(* Logix 5000 project; controller Amvex_Thorpe_Flowmeter vendor 1 type 14 code 106 rev 33.13; software revision 33.01; part 15 of 16 *)
(* tags used below, declared in another part *)
   Auto_Seq : SEQ;
   Clear_TM : TIMER;
   Counter_ONS : BOOL;
   FAULT : DINT;
   FAULTED : DINT;
   Flash_Timer_Off : TIMER;
   Flash_Timer_On : TIMER;
   MODE : MODE;
   RCD_ONS : BOOL;
   RESET : BOOL;
   RESET_ONS : BOOL;
   End_Of_Cycle : BOOL;
   Fitting_Cycle_Timer : TIMER;
   Fitting_Cycle_Timer_DINT : DINT;
   Fitting_Cycle_Timer_ONS : BOOL;
   HMI : HMI_Temp;
   RCP1 : RCP1;
   RCP1_00 : UDT_ID0;
(* RPC1_Main, continued *)

ROUTINE R02_OUTPUTS   (* ladder *)
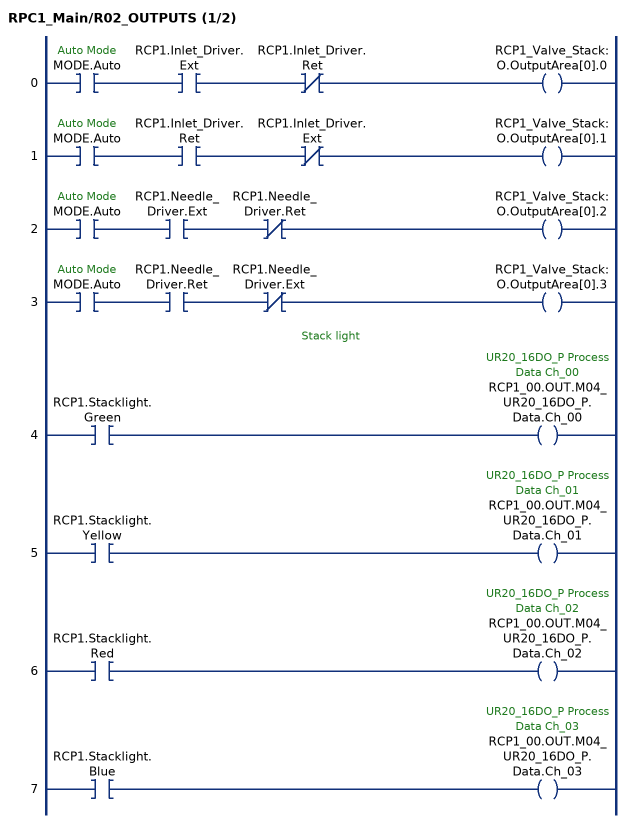
   0: XIC(MODE.Auto)XIC(RCP1.Inlet_Driver.Ext)XIO(RCP1.Inlet_Driver.Ret)OTE(RCP1_Valve_Stack:O.OutputArea[0].0);
   1: XIC(MODE.Auto)XIC(RCP1.Inlet_Driver.Ret)XIO(RCP1.Inlet_Driver.Ext)OTE(RCP1_Valve_Stack:O.OutputArea[0].1);
   2: XIC(MODE.Auto)XIC(RCP1.Needle_Driver.Ext)XIO(RCP1.Needle_Driver.Ret)OTE(RCP1_Valve_Stack:O.OutputArea[0].2);
   3: XIC(MODE.Auto)XIC(RCP1.Needle_Driver.Ret)XIO(RCP1.Needle_Driver.Ext)OTE(RCP1_Valve_Stack:O.OutputArea[0].3);
   // Stack light
   4: XIC(RCP1.Stacklight.Green)OTE(RCP1_00.OUT.M04_UR20_16DO_P.Data.Ch_00);
   5: XIC(RCP1.Stacklight.Yellow)OTE(RCP1_00.OUT.M04_UR20_16DO_P.Data.Ch_01);
   6: XIC(RCP1.Stacklight.Red)OTE(RCP1_00.OUT.M04_UR20_16DO_P.Data.Ch_02);
   7: XIC(RCP1.Stacklight.Blue)OTE(RCP1_00.OUT.M04_UR20_16DO_P.Data.Ch_03);
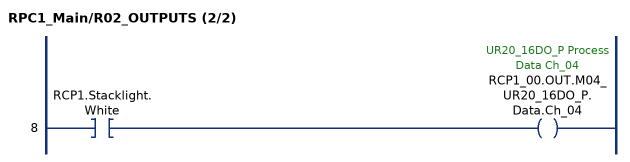
   8: XIC(RCP1.Stacklight.White)OTE(RCP1_00.OUT.M04_UR20_16DO_P.Data.Ch_04);
END_ROUTINE

ROUTINE R03_AUTO_SEQ   (* ladder *)
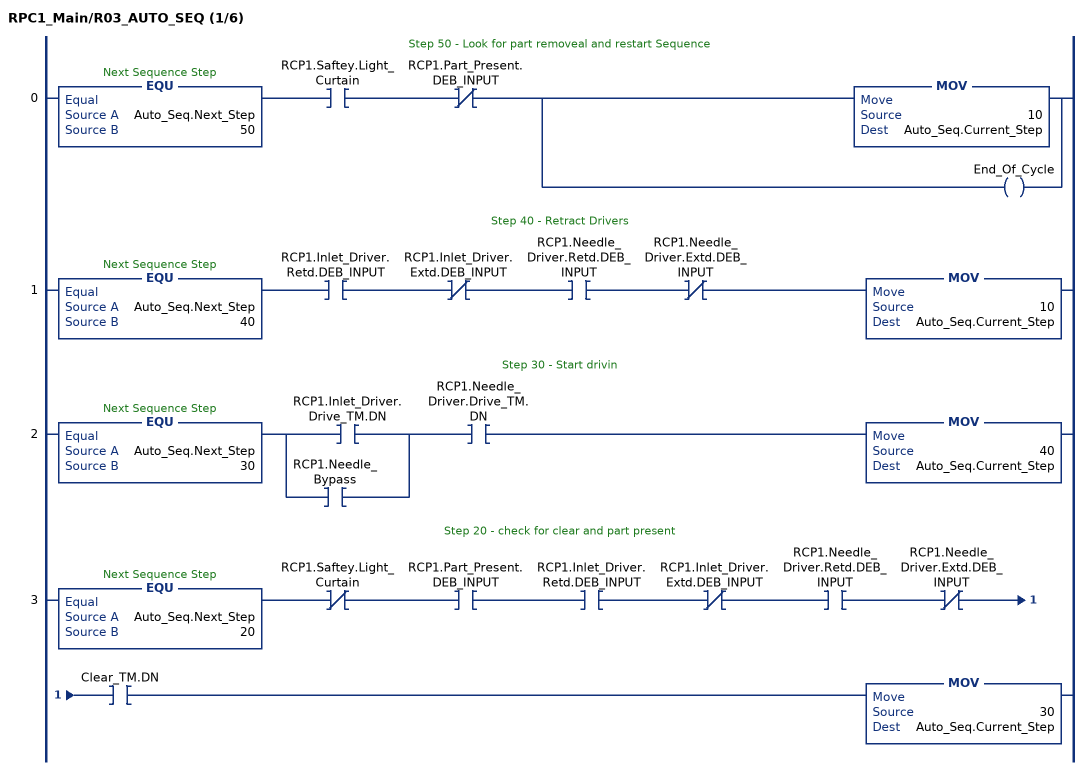
   // Step 50 - Look for part removeal and restart Sequence
   0: EQU(Auto_Seq.Next_Step,50)XIC(RCP1.Saftey.Light_Curtain)XIO(RCP1.Part_Present.DEB_INPUT)[MOV(10,Auto_Seq.Current_Step) ,OTE(End_Of_Cycle) ];
   // Step 40 - Retract Drivers
   1: EQU(Auto_Seq.Next_Step,40)XIC(RCP1.Inlet_Driver.Retd.DEB_INPUT)XIO(RCP1.Inlet_Driver.Extd.DEB_INPUT)XIC(RCP1.Needle_Driver.Retd.DEB_INPUT)XIO(RCP1.Needle_Driver.Extd.DEB_INPUT)MOV(10,Auto_Seq.Current_Step);
   // Step 30 - Start drivin
   2: EQU(Auto_Seq.Next_Step,30)[XIC(RCP1.Inlet_Driver.Drive_TM.DN) ,XIC(RCP1.Needle_Bypass) ]XIC(RCP1.Needle_Driver.Drive_TM.DN)MOV(40,Auto_Seq.Current_Step);
   // Step 20 - check for clear and part present
   3: EQU(Auto_Seq.Next_Step,20)XIO(RCP1.Saftey.Light_Curtain)XIC(RCP1.Part_Present.DEB_INPUT)XIC(RCP1.Inlet_Driver.Retd.DEB_INPUT)XIO(RCP1.Inlet_Driver.Extd.DEB_INPUT)XIC(RCP1.Needle_Driver.Retd.DEB_INPUT)XIO(RCP1.Needle_Driver.Extd.DEB_INPUT)XIC(Clear_TM.DN)MOV(30,Auto_Seq.Current_Step);
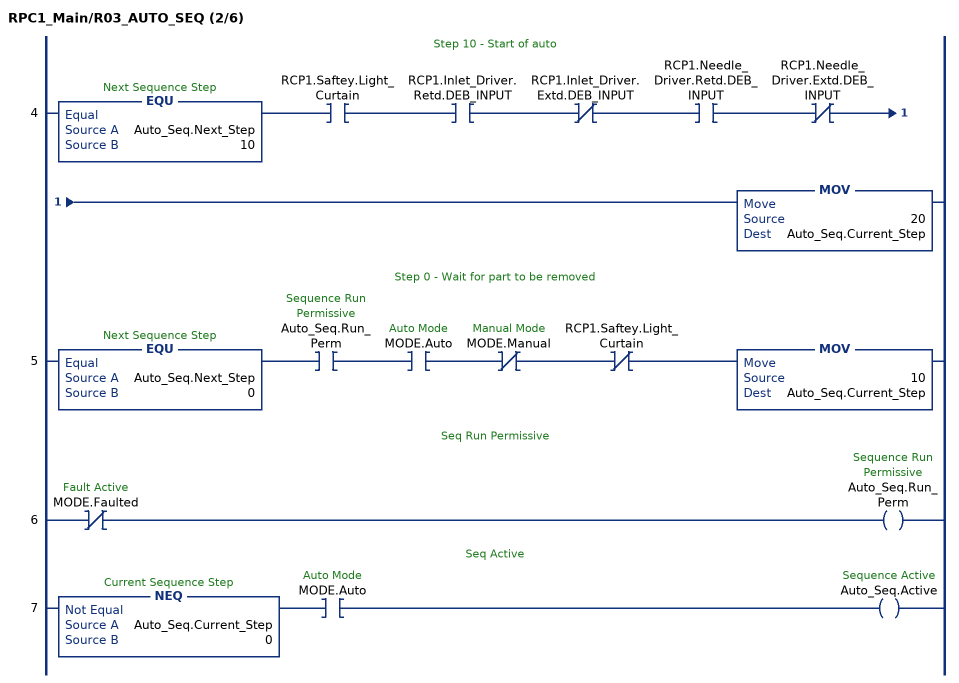
   // Step 10 - Start of auto
   4: EQU(Auto_Seq.Next_Step,10)XIC(RCP1.Saftey.Light_Curtain)XIC(RCP1.Inlet_Driver.Retd.DEB_INPUT)XIO(RCP1.Inlet_Driver.Extd.DEB_INPUT)XIC(RCP1.Needle_Driver.Retd.DEB_INPUT)XIO(RCP1.Needle_Driver.Extd.DEB_INPUT)MOV(20,Auto_Seq.Current_Step);
   // Step 0 - Wait for part to be removed
   5: EQU(Auto_Seq.Next_Step,0)XIC(Auto_Seq.Run_Perm)XIC(MODE.Auto)XIO(MODE.Manual)XIO(RCP1.Saftey.Light_Curtain)MOV(10,Auto_Seq.Current_Step);
   // Seq Run Permissive
   6: XIO(MODE.Faulted)OTE(Auto_Seq.Run_Perm);
   // Seq Active
   7: NEQ(Auto_Seq.Current_Step,0)XIC(MODE.Auto)OTE(Auto_Seq.Active);
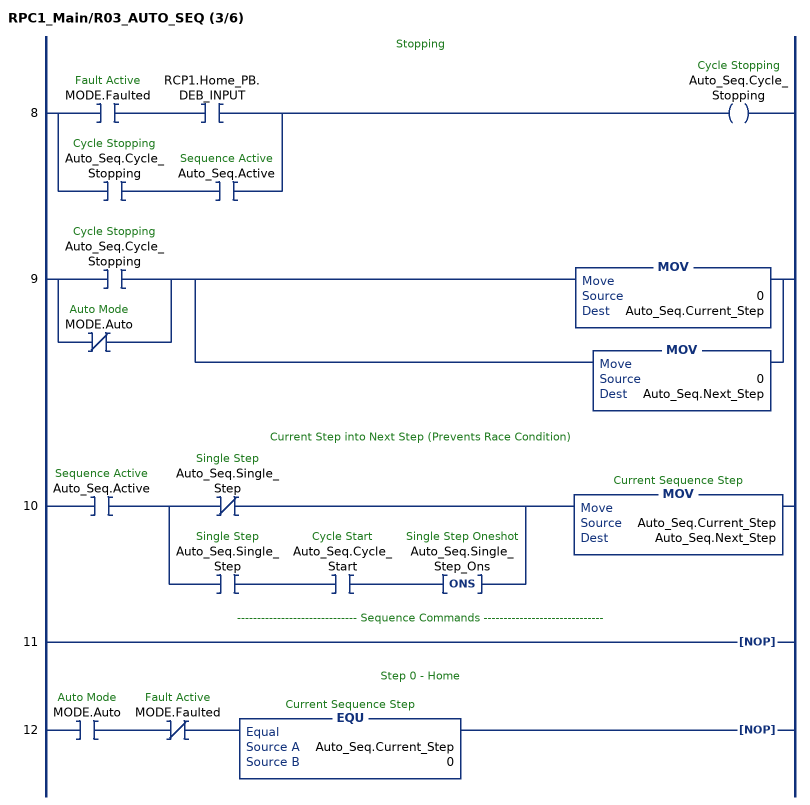
   // Stopping
   8: [XIC(MODE.Faulted) XIC(RCP1.Home_PB.DEB_INPUT) ,XIC(Auto_Seq.Cycle_Stopping) XIC(Auto_Seq.Active) ]OTE(Auto_Seq.Cycle_Stopping);
   9: [XIC(Auto_Seq.Cycle_Stopping) ,XIO(MODE.Auto) ][MOV(0,Auto_Seq.Current_Step) ,MOV(0,Auto_Seq.Next_Step) ];
   // Current Step into Next Step (Prevents Race Condition)
   10: XIC(Auto_Seq.Active)[XIO(Auto_Seq.Single_Step) ,XIC(Auto_Seq.Single_Step) XIC(Auto_Seq.Cycle_Start) ONS(Auto_Seq.Single_Step_Ons) ]MOV(Auto_Seq.Current_Step,Auto_Seq.Next_Step);
   // ------------------------------ Sequence Commands ------------------------------
   11: NOP();
   // Step 0 - Home
   12: XIC(MODE.Auto)XIO(MODE.Faulted)EQU(Auto_Seq.Current_Step,0)NOP();
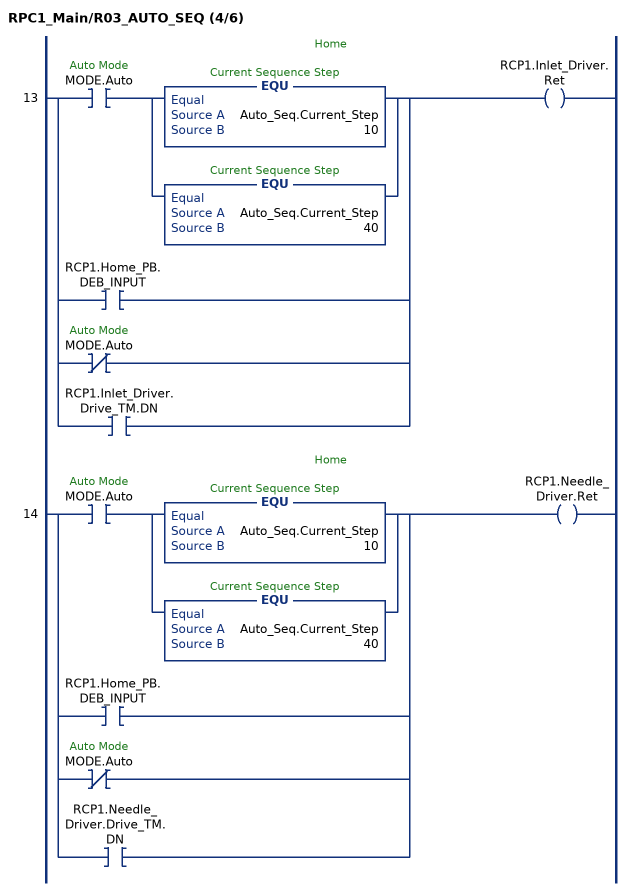
   // Home
   13: [XIC(MODE.Auto) [EQU(Auto_Seq.Current_Step,10) ,EQU(Auto_Seq.Current_Step,40) ] ,XIC(RCP1.Home_PB.DEB_INPUT) ,XIO(MODE.Auto) ,XIC(RCP1.Inlet_Driver.Drive_TM.DN) ]OTE(RCP1.Inlet_Driver.Ret);
   // Home
   14: [XIC(MODE.Auto) [EQU(Auto_Seq.Current_Step,10) ,EQU(Auto_Seq.Current_Step,40) ] ,XIC(RCP1.Home_PB.DEB_INPUT) ,XIO(MODE.Auto) ,XIC(RCP1.Needle_Driver.Drive_TM.DN) ]OTE(RCP1.Needle_Driver.Ret);
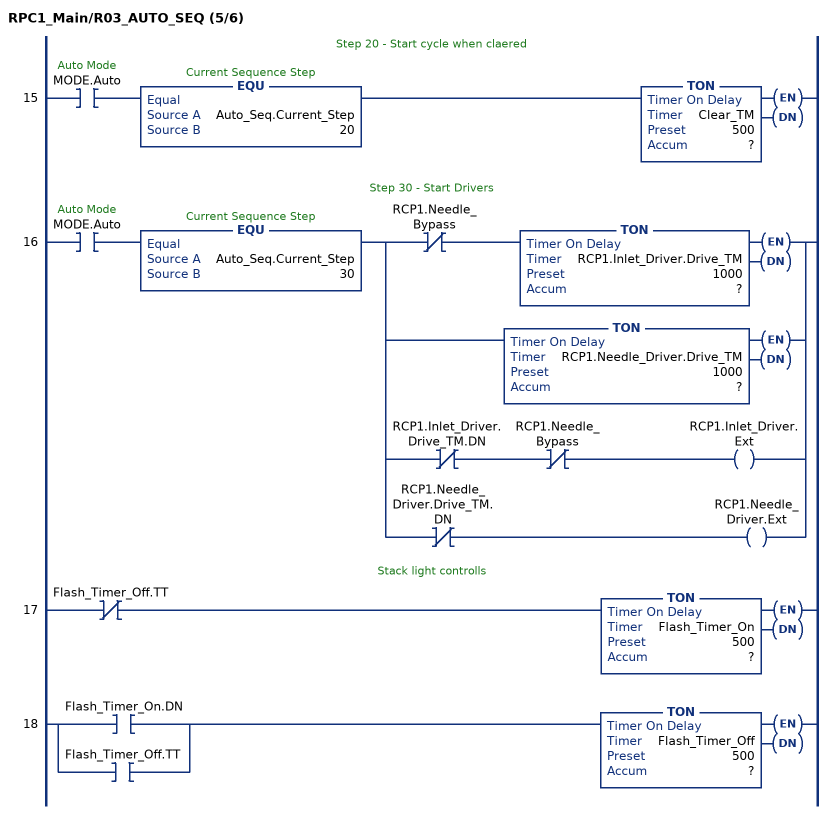
   // Step 20 - Start cycle when claered
   15: XIC(MODE.Auto)EQU(Auto_Seq.Current_Step,20)TON(Clear_TM,?,?);
   // Step 30 - Start Drivers
   16: XIC(MODE.Auto)EQU(Auto_Seq.Current_Step,30)[XIO(RCP1.Needle_Bypass) TON(RCP1.Inlet_Driver.Drive_TM,?,?) ,TON(RCP1.Needle_Driver.Drive_TM,?,?) ,XIO(RCP1.Inlet_Driver.Drive_TM.DN) XIO(RCP1.Needle_Bypass) OTE(RCP1.Inlet_Driver.Ext) ,XIO(RCP1.Needle_Driver.Drive_TM.DN) OTE(RCP1.Needle_Driver.Ext) ];
   // Stack light controlls
   17: XIO(Flash_Timer_Off.TT)TON(Flash_Timer_On,?,?);
   18: [XIC(Flash_Timer_On.DN) ,XIC(Flash_Timer_Off.TT) ]TON(Flash_Timer_Off,?,?);
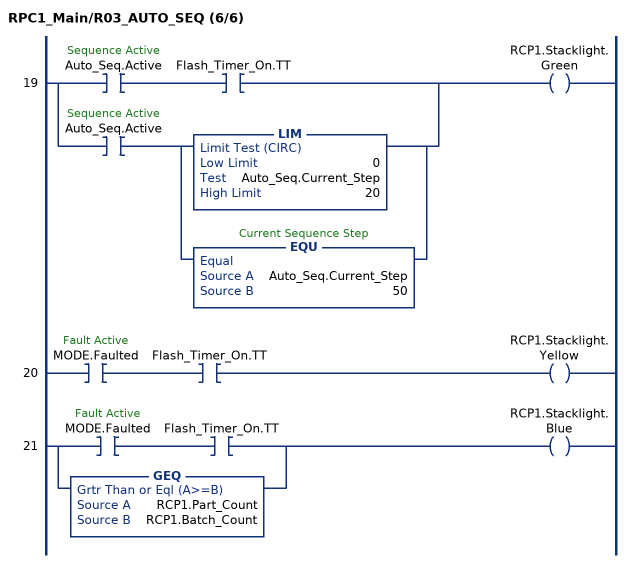
   19: [XIC(Auto_Seq.Active) XIC(Flash_Timer_On.TT) ,XIC(Auto_Seq.Active) [LIM(0,Auto_Seq.Current_Step,20) ,EQU(Auto_Seq.Current_Step,50) ] ]OTE(RCP1.Stacklight.Green);
   20: XIC(MODE.Faulted)XIC(Flash_Timer_On.TT)OTE(RCP1.Stacklight.Yellow);
   21: [XIC(MODE.Faulted) XIC(Flash_Timer_On.TT) ,GEQ(RCP1.Part_Count,RCP1.Batch_Count) ]OTE(RCP1.Stacklight.Blue);
END_ROUTINE

ROUTINE R04_FAULTS   (* ladder *)
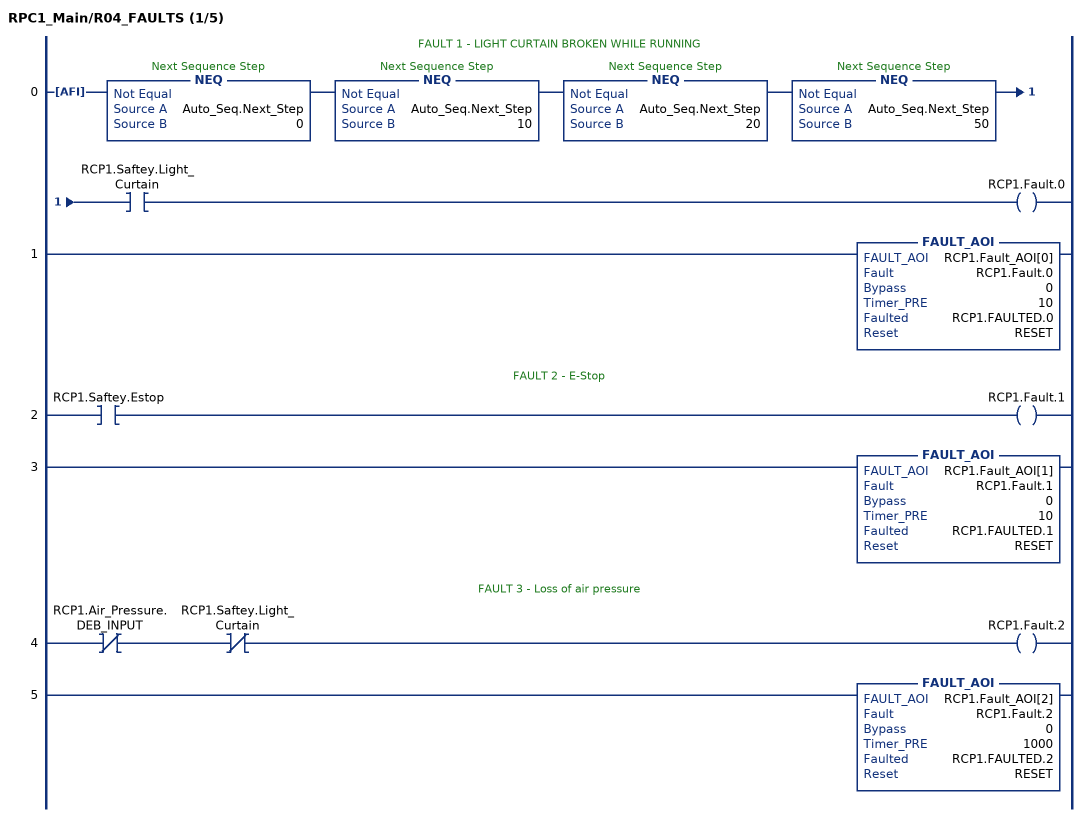
   // FAULT 1 - LIGHT CURTAIN BROKEN WHILE RUNNING
   0: AFI()NEQ(Auto_Seq.Next_Step,0)NEQ(Auto_Seq.Next_Step,10)NEQ(Auto_Seq.Next_Step,20)NEQ(Auto_Seq.Next_Step,50)XIC(RCP1.Saftey.Light_Curtain)OTE(RCP1.Fault.0);
   1: FAULT_AOI(RCP1.Fault_AOI[0],RCP1.Fault.0,0,10,RCP1.FAULTED.0,RESET);
   // FAULT 2 - E-Stop
   2: XIC(RCP1.Saftey.Estop)OTE(RCP1.Fault.1);
   3: FAULT_AOI(RCP1.Fault_AOI[1],RCP1.Fault.1,0,10,RCP1.FAULTED.1,RESET);
   // FAULT 3 - Loss of air pressure
   4: XIO(RCP1.Air_Pressure.DEB_INPUT)XIO(RCP1.Saftey.Light_Curtain)OTE(RCP1.Fault.2);
   5: FAULT_AOI(RCP1.Fault_AOI[2],RCP1.Fault.2,0,1000,RCP1.FAULTED.2,RESET);
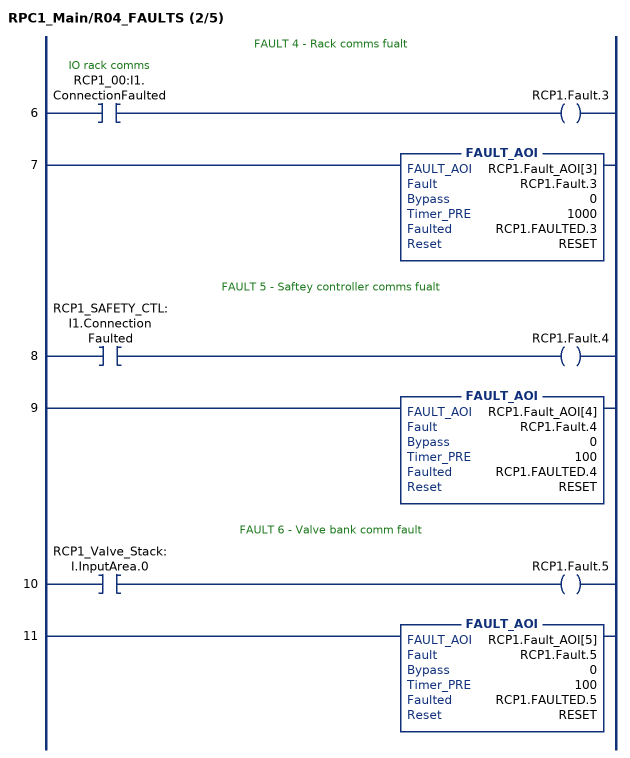
   // FAULT 4 - Rack comms fualt
   6: XIC(RCP1_00:I1.ConnectionFaulted)OTE(RCP1.Fault.3);
   7: FAULT_AOI(RCP1.Fault_AOI[3],RCP1.Fault.3,0,1000,RCP1.FAULTED.3,RESET);
   // FAULT 5 - Saftey controller comms fualt
   8: XIC(RCP1_SAFETY_CTL:I1.ConnectionFaulted)OTE(RCP1.Fault.4);
   9: FAULT_AOI(RCP1.Fault_AOI[4],RCP1.Fault.4,0,100,RCP1.FAULTED.4,RESET);
   // FAULT 6 - Valve bank comm fault
   10: XIC(RCP1_Valve_Stack:I.InputArea.0)OTE(RCP1.Fault.5);
   11: FAULT_AOI(RCP1.Fault_AOI[5],RCP1.Fault.5,0,100,RCP1.FAULTED.5,RESET);
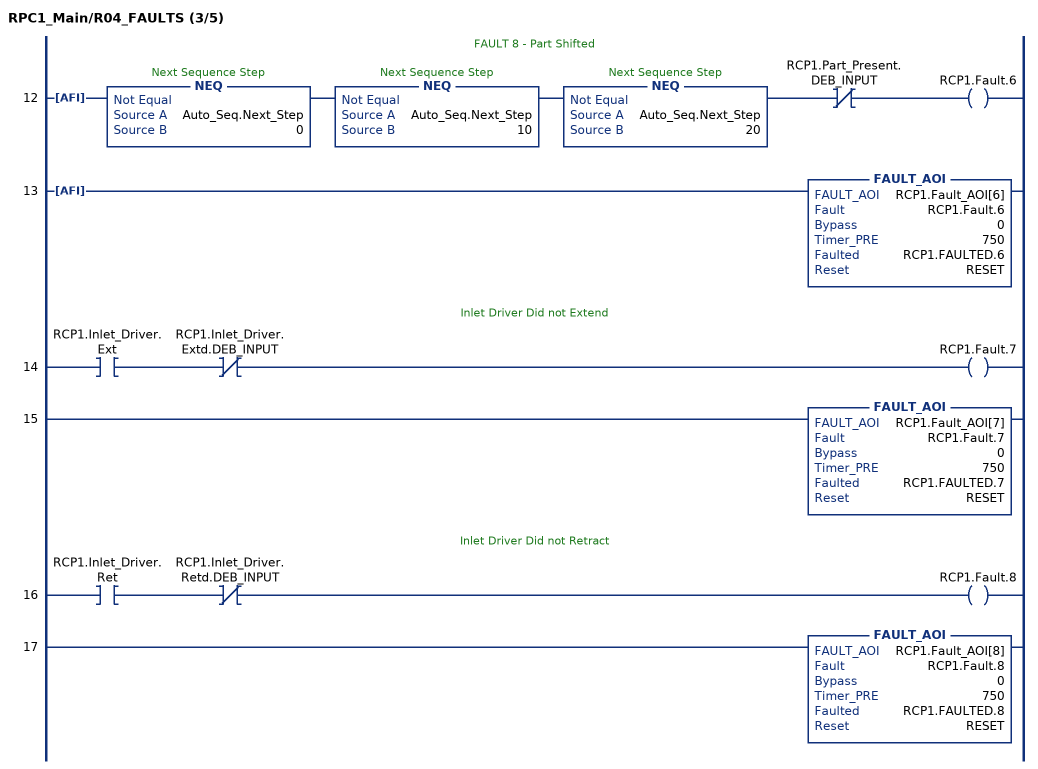
   // FAULT 8 - Part Shifted
   12: AFI()NEQ(Auto_Seq.Next_Step,0)NEQ(Auto_Seq.Next_Step,10)NEQ(Auto_Seq.Next_Step,20)XIO(RCP1.Part_Present.DEB_INPUT)OTE(RCP1.Fault.6);
   13: AFI()FAULT_AOI(RCP1.Fault_AOI[6],RCP1.Fault.6,0,750,RCP1.FAULTED.6,RESET);
   // Inlet Driver Did not Extend
   14: XIC(RCP1.Inlet_Driver.Ext)XIO(RCP1.Inlet_Driver.Extd.DEB_INPUT)OTE(RCP1.Fault.7);
   15: FAULT_AOI(RCP1.Fault_AOI[7],RCP1.Fault.7,0,750,RCP1.FAULTED.7,RESET);
   // Inlet Driver Did not Retract
   16: XIC(RCP1.Inlet_Driver.Ret)XIO(RCP1.Inlet_Driver.Retd.DEB_INPUT)OTE(RCP1.Fault.8);
   17: FAULT_AOI(RCP1.Fault_AOI[8],RCP1.Fault.8,0,750,RCP1.FAULTED.8,RESET);
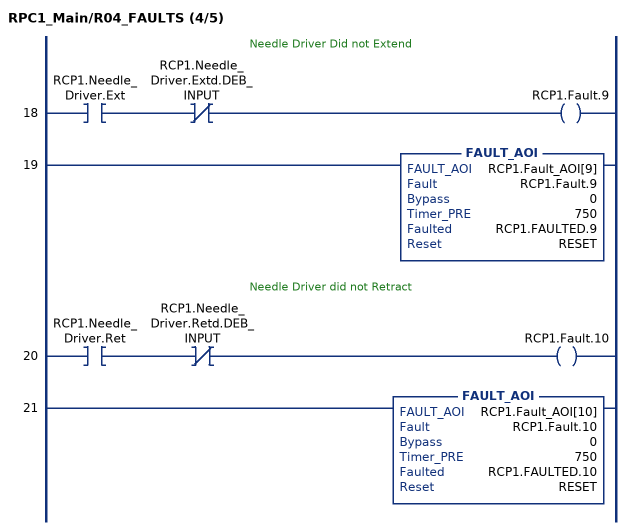
   // Needle Driver Did not Extend
   18: XIC(RCP1.Needle_Driver.Ext)XIO(RCP1.Needle_Driver.Extd.DEB_INPUT)OTE(RCP1.Fault.9);
   19: FAULT_AOI(RCP1.Fault_AOI[9],RCP1.Fault.9,0,750,RCP1.FAULTED.9,RESET);
   // Needle Driver did not Retract
   20: XIC(RCP1.Needle_Driver.Ret)XIO(RCP1.Needle_Driver.Retd.DEB_INPUT)OTE(RCP1.Fault.10);
   21: FAULT_AOI(RCP1.Fault_AOI[10],RCP1.Fault.10,0,750,RCP1.FAULTED.10,RESET);
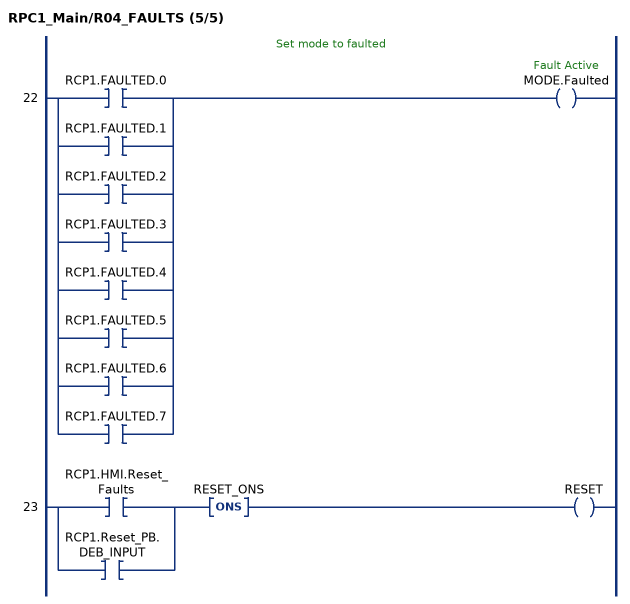
   // Set mode to faulted
   22: [XIC(RCP1.FAULTED.0) ,XIC(RCP1.FAULTED.1) ,XIC(RCP1.FAULTED.2) ,XIC(RCP1.FAULTED.3) ,XIC(RCP1.FAULTED.4) ,XIC(RCP1.FAULTED.5) ,XIC(RCP1.FAULTED.6) ,XIC(RCP1.FAULTED.7) ]OTE(MODE.Faulted);
   23: [XIC(RCP1.HMI.Reset_Faults) ,XIC(RCP1.Reset_PB.DEB_INPUT) ]ONS(RESET_ONS)OTE(RESET);
END_ROUTINE

ROUTINE R05_SAFETY_CONTROLLER   (* ladder *)
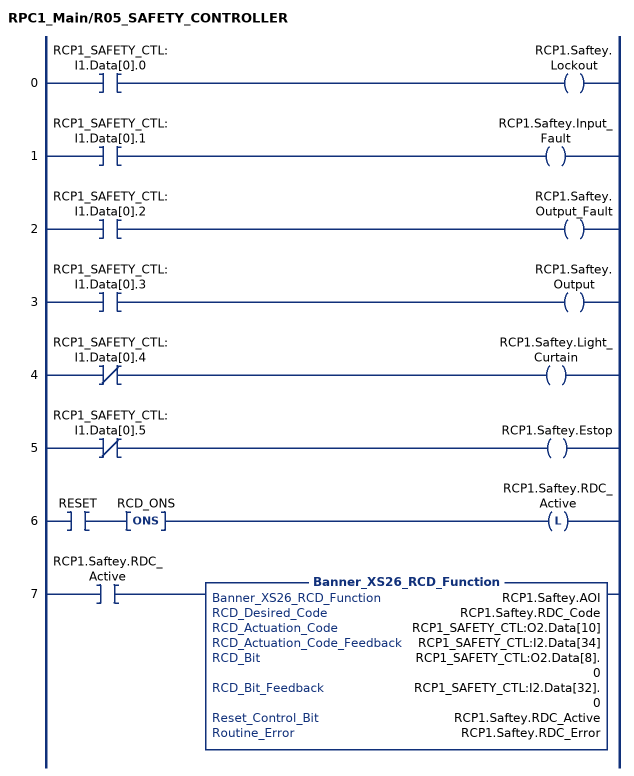
   0: XIC(RCP1_SAFETY_CTL:I1.Data[0].0)OTE(RCP1.Saftey.Lockout);
   1: XIC(RCP1_SAFETY_CTL:I1.Data[0].1)OTE(RCP1.Saftey.Input_Fault);
   2: XIC(RCP1_SAFETY_CTL:I1.Data[0].2)OTE(RCP1.Saftey.Output_Fault);
   3: XIC(RCP1_SAFETY_CTL:I1.Data[0].3)OTE(RCP1.Saftey.Output);
   4: XIO(RCP1_SAFETY_CTL:I1.Data[0].4)OTE(RCP1.Saftey.Light_Curtain);
   5: XIO(RCP1_SAFETY_CTL:I1.Data[0].5)OTE(RCP1.Saftey.Estop);
   6: XIC(RESET)ONS(RCD_ONS)OTL(RCP1.Saftey.RDC_Active);
   7: XIC(RCP1.Saftey.RDC_Active)Banner_XS26_RCD_Function(RCP1.Saftey.AOI,RCP1.Saftey.RDC_Code,RCP1_SAFETY_CTL:O2.Data[10],RCP1_SAFETY_CTL:I2.Data[34],RCP1_SAFETY_CTL:O2.Data[8].0,RCP1_SAFETY_CTL:I2.Data[32].0,RCP1.Saftey.RDC_Active,RCP1.Saftey.RDC_Error);
END_ROUTINE

ROUTINE R06_HMI   (* ladder *)
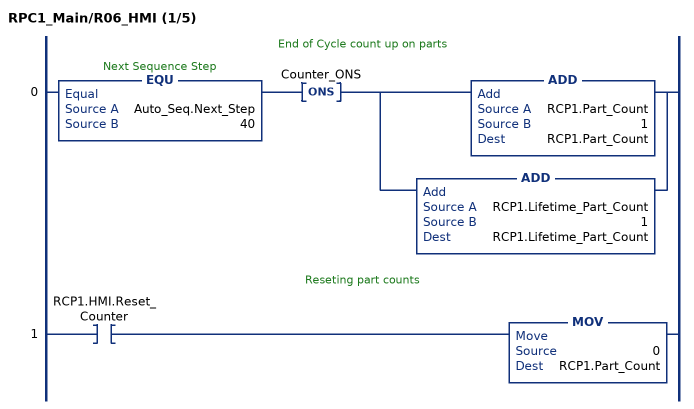
   // End of Cycle count up on parts
   0: EQU(Auto_Seq.Next_Step,40)ONS(Counter_ONS)[ADD(RCP1.Part_Count,1,RCP1.Part_Count) ,ADD(RCP1.Lifetime_Part_Count,1,RCP1.Lifetime_Part_Count) ];
   // Reseting part counts
   1: XIC(RCP1.HMI.Reset_Counter)MOV(0,RCP1.Part_Count);
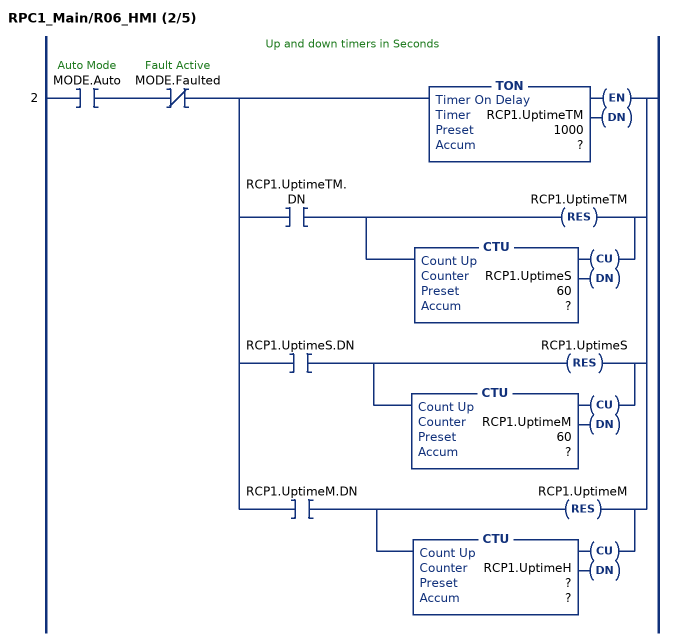
   // Up and down timers in Seconds
   2: XIC(MODE.Auto)XIO(MODE.Faulted)[TON(RCP1.UptimeTM,?,?) ,XIC(RCP1.UptimeTM.DN) [RES(RCP1.UptimeTM) ,CTU(RCP1.UptimeS,?,?) ] ,XIC(RCP1.UptimeS.DN) [RES(RCP1.UptimeS) ,CTU(RCP1.UptimeM,?,?) ] ,XIC(RCP1.UptimeM.DN) [RES(RCP1.UptimeM) ,CTU(RCP1.UptimeH,?,?) ] ];
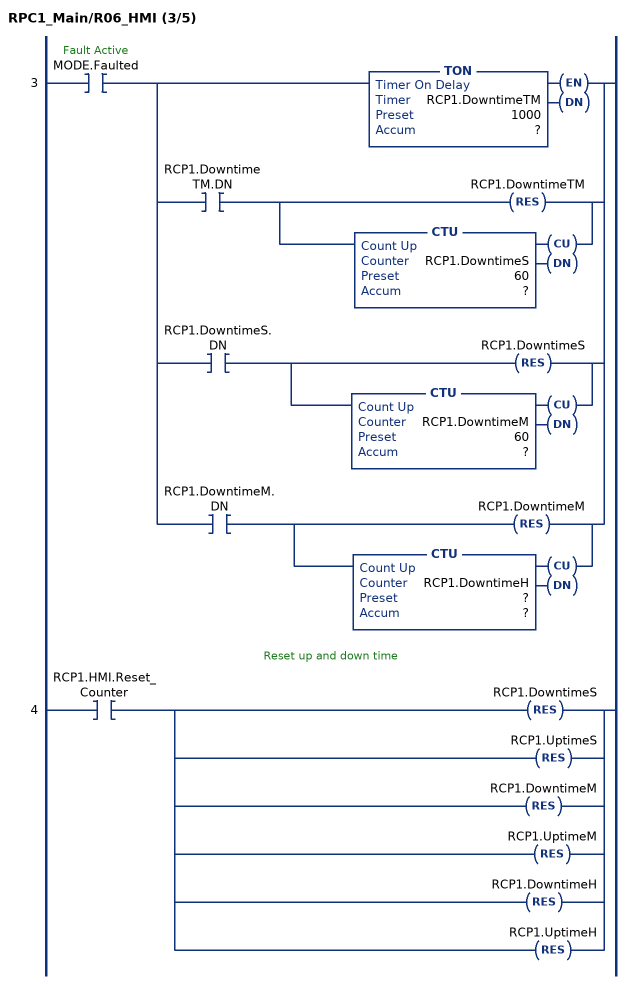
   3: XIC(MODE.Faulted)[TON(RCP1.DowntimeTM,?,?) ,XIC(RCP1.DowntimeTM.DN) [RES(RCP1.DowntimeTM) ,CTU(RCP1.DowntimeS,?,?) ] ,XIC(RCP1.DowntimeS.DN) [RES(RCP1.DowntimeS) ,CTU(RCP1.DowntimeM,?,?) ] ,XIC(RCP1.DowntimeM.DN) [RES(RCP1.DowntimeM) ,CTU(RCP1.DowntimeH,?,?) ] ];
   // Reset up and down time
   4: XIC(RCP1.HMI.Reset_Counter)[RES(RCP1.DowntimeS) ,RES(RCP1.UptimeS) ,RES(RCP1.DowntimeM) ,RES(RCP1.UptimeM) ,RES(RCP1.DowntimeH) ,RES(RCP1.UptimeH) ];
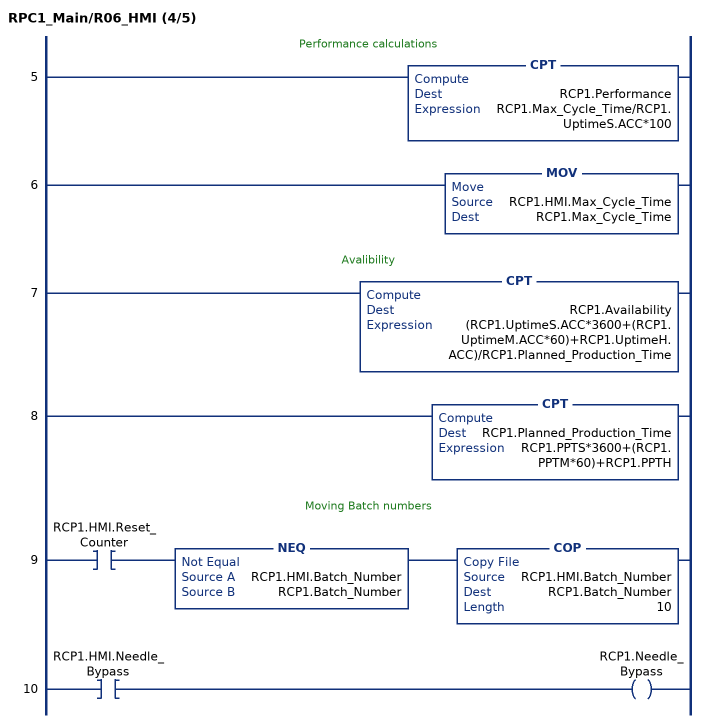
   // Performance calculations
   5: CPT(RCP1.Performance,RCP1.Max_Cycle_Time/RCP1.UptimeS.ACC*100);
   6: MOV(RCP1.HMI.Max_Cycle_Time,RCP1.Max_Cycle_Time);
   // Avalibility
   7: CPT(RCP1.Availability,(RCP1.UptimeS.ACC*3600+(RCP1.UptimeM.ACC*60)+RCP1.UptimeH.ACC)/RCP1.Planned_Production_Time);
   8: CPT(RCP1.Planned_Production_Time,RCP1.PPTS*3600+(RCP1.PPTM*60)+RCP1.PPTH);
   // Moving Batch numbers
   9: XIC(RCP1.HMI.Reset_Counter)NEQ(RCP1.HMI.Batch_Number,RCP1.Batch_Number)COP(RCP1.HMI.Batch_Number,RCP1.Batch_Number,10);
   10: XIC(RCP1.HMI.Needle_Bypass)OTE(RCP1.Needle_Bypass);
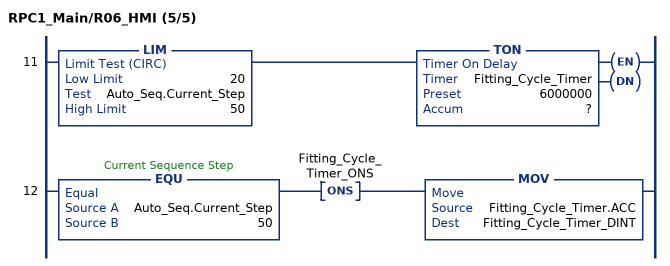
   11: LIM(20,Auto_Seq.Current_Step,50)TON(Fitting_Cycle_Timer,?,?);
   12: EQU(Auto_Seq.Current_Step,50)ONS(Fitting_Cycle_Timer_ONS)MOV(Fitting_Cycle_Timer.ACC,Fitting_Cycle_Timer_DINT);
END_ROUTINE
